{attribute 'qualified_only'}
VAR_GLOBAL CONSTANT
    // Encoder reference values in counts = nm
    // Enc Ref Vals from FAT
    nYUP_ENC_REF : ULINT := 108743550;
    nYDWN_ENC_REF : ULINT := 108243370;
    nXUP_ENC_REF : ULINT := 19628100;
    nXDWN_ENC_REF : ULINT := 20865800;
END_VAR

(* stored: Version 1.1.0.1, ProductVersion 3.1.4022.18
   GVL GVL_M1K3_Constants: Id {e75b3be9-127e-46b4-b219-470b94c00321} *)
